(* IEC 61131-3 sources: actuators/src/notification-service/errors, 3 files *)

(* ---- error.st ---- *)
NAMESPACE NotificationService
    NAMESPACE ErrorHandling
        // Basis Fehlertyp
        TYPE Alarm :
            STRUCT
                id : STRING;
                messageSeverity : Severity;
                source : STRING;
                errorMessage : STRING;
                timestamp : DATE_AND_TIME;
            END_STRUCT;

            Severity : (Info, Warning, Error);
        END_TYPE
    END_NAMESPACE

END_NAMESPACE

(* ---- error-logger.st ---- *)
USING System.Strings;
USING System.Math;
USING NotificationService.Interfaces;

NAMESPACE NotificationService
    NAMESPACE ErrorHandling
        CLASS ErrorLogger IMPLEMENTS ILogger
            VAR CONSTANT
                LOW_ARR_BOUND : INT := 1;
                UP_ARR_BOUND : INT := 12;
            END_VAR

            VAR PROTECTED
                _messages : ARRAY[LOW_ARR_BOUND..UP_ARR_BOUND] OF Alarm;
                _currentFreeIndex : INT := LOW_ARR_BOUND;
            END_VAR

            METHOD PUBLIC Log
                VAR_INPUT
                    e : Alarm;
                END_VAR
                _messages[_currentFreeIndex] := e;
                _currentFreeIndex := _currentFreeIndex + 1;

                IF _currentFreeIndex > UP_ARR_BOUND THEN
                    _currentFreeIndex := LOW_ARR_BOUND;
                END_IF;
            END_METHOD

            METHOD PUBLIC GetLatestAlarms
                VAR_INPUT
                    severityFilter : Severity;
                END_VAR
                VAR_IN_OUT
                    messages : ARRAY[*] OF Alarm;
                END_VAR
                VAR_TEMP
                    requiredMessagesCount, availableMessagesCount : INT;
                    targetIndex, sourceIndex, transferCount : INT;
                    i : INT;
                END_VAR

                requiredMessagesCount := TO_INT(UPPER_BOUND(messages, 1) - LOWER_BOUND(messages, 1)) + 1;
                availableMessagesCount := UP_ARR_BOUND - LOW_ARR_BOUND + 1;

                // calculate the source index from which to start
                sourceIndex := _currentFreeIndex - 1;
                IF sourceIndex < LOW_ARR_BOUND THEN
                    sourceIndex := UP_ARR_BOUND;
                END_IF;

                IF _currentFreeIndex > LOW_ARR_BOUND THEN
                    availableMessagesCount := _currentFreeIndex - LOW_ARR_BOUND;
               END_IF;

                // determine the minimum possible amount of messages to be transfered
                transferCount := Min(requiredMessagesCount, availableMessagesCount);

                // Copy messages, starting from the newest
                FOR i := 0 TO transferCount - 1 DO
                    targetIndex := TO_INT(LOWER_BOUND(messages, 1)) + i;

                    messages[targetIndex] := _messages[sourceIndex];

                    sourceIndex := sourceIndex - 1;
                    IF sourceIndex < LOW_ARR_BOUND THEN
                        sourceIndex := UP_ARR_BOUND;
                    END_IF;
                END_FOR;
            END_METHOD
        END_CLASS
    END_NAMESPACE
END_NAMESPACE

(* ---- error-provider-base.st ---- *)
USING System.Strings;
USING NotificationService.Interfaces;
USING Simatic.Ax.Commands;

NAMESPACE NotificationService
    NAMESPACE ErrorHandling
        CLASS ErrorProviderBase IMPLEMENTS IAlarmProvider
            VAR PUBLIC
                _id : STRING;
                _name : STRING;

            END_VAR

            VAR PUBLIC
                _notificationService : INotificationService;
            END_VAR

            METHOD PUBLIC SetNotificationService
                VAR_INPUT
                    ns : INotificationService;
                END_VAR
                _notificationService := ns;
            END_METHOD

            METHOD PUBLIC Notify : BOOL
                VAR_INPUT
                    e : Alarm;
                END_VAR

                VAR_TEMP
                    t : Alarm;
                END_VAR
                t := e;
                IF e.source = '' THEN
                    t.source := _name;
                ELSE
                    t.source := Concat(_name, '.', e.source);
                END_IF;
                _notificationService.RegisterAlarm(THIS, t);
                THIS.OnNotification();
                Notify := TRUE;
            END_METHOD

            METHOD PUBLIC OnNotification ; END_METHOD

            // // concatenation of bools incorrect
            // METHOD PUBLIC Notify : BOOL
            //     VAR_INPUT
            //         errors : ARRAY[*] OF Alarm;
            //     END_VAR
            //     VAR_TEMP
            //         i, j : DINT := 0;
            //         result : BOOL := FALSE;
            //     END_VAR
            //     i := LOWER_BOUND(errors, 1);
            //     j := UPPER_BOUND(errors, 1);

            //     FOR i := LOWER_BOUND(errors, 1) TO UPPER_BOUND(errors, 1) DO
            //         result := _notificationService.RegisterAlarm(THIS, errors[i]);
            //     END_FOR;

            //     THIS.OnNotification();

            //     Notify := result;
            // END_METHOD

            METHOD PUBLIC Equals : BOOL
                VAR_INPUT
                    other : IComparable;
                END_VAR
                VAR
                    i : REF_TO ErrorProviderBase;
                END_VAR
                IF other = NULL THEN
                    Equals := FALSE;
                    RETURN;
                END_IF;
                i ?= other;

                IF i = NULL THEN
                    Equals := FALSE;
                    RETURN;
                END_IF;

                IF i^._id <> _id THEN
                    Equals := FALSE;
                    RETURN;
                END_IF;
                Equals := TRUE;

            END_METHOD

            // just here for the ease of spawning an error
            METHOD PUBLIC Execute
                VAR_INPUT
                    triggerError : BOOL;
                    message : STRING;
                    timestamp : DATE_AND_TIME;
                    sev : Severity;
                END_VAR
                VAR_TEMP
                    e : Alarm;
                END_VAR

                IF triggerError THEN
                    e.errorMessage := message;
                    e.timestamp := timestamp;
                    e.messageSeverity := sev;
                    THIS.Notify(e);
                END_IF;
            END_METHOD
        END_CLASS
    END_NAMESPACE
END_NAMESPACE
